(* PLC project SafeLOGIC-1, BrAutomation SafeDESIGNER  4.4.0.0 *)
(* stored: companyURL http://www.br-automation.com, creationDateTime Thu Mar 18 11:06:18 2021 *)

PROGRAM Main

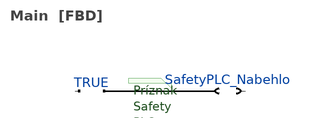
(* FBD diagram, written out as Structured Text *)
(* Príznak Safety PLC nabehlo *)
SafetyPLC_Nabehlo := TRUE;
END_PROGRAM
